INTERFACE I_Animation

PROPERTY PUBLIC CurrentFrameImage : ITcVnImage
GET
END_GET
END_PROPERTY

PROPERTY PUBLIC CurrentFrameIndex : UDINT
GET
END_GET
END_PROPERTY

PROPERTY PUBLIC IsAtLastFrame : BOOL
GET
END_GET
END_PROPERTY

METHOD PUBLIC MoveToStart
VAR_INPUT
END_VAR
END_METHOD

PROPERTY PUBLIC TotalFrameCount : UDINT
GET
END_GET
END_PROPERTY

METHOD PUBLIC TryMoveNext : BOOL
VAR_INPUT
END_VAR
END_METHOD

METHOD PUBLIC TryMovePrevious : BOOL
VAR_INPUT
END_VAR
END_METHOD

END_INTERFACE

(* stored: Version 1.1.0.1, ProductVersion 3.1.4024.13
   Itf I_Animation: Id {20dcdc20-ac32-492a-b601-1441e2deba44}
   Property CurrentFrameImage: Id {e24c7b4e-7a71-4359-b239-1442fc999968}
   Get Get: Id {602f10dc-c391-4daf-becd-d9115a8a96f6}
   Property CurrentFrameIndex: Id {53cab9b4-1932-453a-afe7-fc7cc17ac78f}
   Get Get: Id {930f5b1b-b15e-4210-9722-cfc0c12ff03b}
   Property IsAtLastFrame: Id {b15b8093-fe91-4059-b3da-e93cce440d9f}
   Get Get: Id {f53b825a-453a-4869-9bef-0e86731871e5}
   Method MoveToStart: Id {5c008f78-422d-4a7f-a63d-1603de9ef052}
   Property TotalFrameCount: Id {3b4e34b7-e50d-452b-8e69-f5e9639d6366}
   Get Get: Id {90105280-94cf-4060-85a0-ed85bf9b298b}
   Method TryMoveNext: Id {5b3a2899-139f-4b18-9dbd-293e969b8679}
   Method TryMovePrevious: Id {e2f36904-72a2-455f-a2e3-97c9d49193c5} *)
